// TIA Portal project "双流水线程序控制" (V16)

(* hardware
DEVICE "S7-1200 station_1"  S7-1200 Station
   slot 0: "Rack_0"  S7-1200 Rack  Rack  V1.0
   slot 1: "PLC_1"  CPU 1214C DC/DC/Rly  6ES7 214-1HG40-0XB0  V4.4
*)

// ===== PLC "PLC_1"  CPU 1214C DC/DC/Rly =====

VAR_GLOBAL   // PLC tag table "默认变量表"
   "Tag_1" AT %M1.0 : Bool;
   "Tag_2" AT %M1.1 : Bool;
END_VAR

VAR_GLOBAL   // PLC tag table "io表"
   "传感器9" AT %I0.0 : Bool;
   "传感器8" AT %I0.1 : Bool;
   "传感器7" AT %I0.2 : Bool;
   "传感器1" AT %I0.3 : Bool;
   "传感器2" AT %I0.4 : Bool;
   "传感器3" AT %I0.5 : Bool;
   "传感器4" AT %I0.6 : Bool;
   "传感器5" AT %I0.7 : Bool;
   "传感器6" AT %I1.0 : Bool;
   "传感器10" AT %I1.1 : Bool;
   "开始" AT %I1.2 : Bool;
   "复位" AT %I1.3 : Bool;
   "停止" AT %I1.4 : Bool;
   "紧急停止" AT %I1.5 : Bool;
   "1挡" AT %I1.6 : Bool;
   "FACTORY I/O (Running)" AT %I1.7 : Bool;
   "前后" AT %Q0.0 : Bool;
   "上下" AT %Q0.1 : Bool;
   "吸取" AT %Q0.2 : Bool;
   "皮带1" AT %Q0.3 : Bool;
   "推上盖" AT %Q0.4 : Bool;
   "上升1" AT %Q0.5 : Bool;
   "皮带2" AT %Q0.6 : Bool;
   "推下盖" AT %Q0.7 : Bool;
   "上升2" AT %Q1.0 : Bool;
   "绿灯" AT %Q1.1 : Bool;
   "黄灯" AT %Q1.2 : Bool;
   "红灯" AT %Q1.3 : Bool;
   "显示屏" AT %QD30 : DInt;
END_VAR

// folder: 02-启动

DATA_BLOCK "启动_DB"   // DB2
{ S7_Optimized_Access := 'TRUE' }
VERSION : 0.1
// stored: InstanceOfName 启动
"启动"
BEGIN
END_DATA_BLOCK

// folder: 02-核心组装区

DATA_BLOCK "核心组装区_DB"   // DB1
{ S7_Optimized_Access := 'TRUE' }
VERSION : 0.1
// stored: InstanceOfName 核心组装区
"核心组装区"
BEGIN
END_DATA_BLOCK

// folder: (top level)

FUNCTION "MHJ-PLC-Lab-Function-S71200" : Void   // FC9000, SCL
{ S7_Optimized_Access := 'TRUE' }
VERSION : 0.1
   VAR_TEMP
      rdTimeReturn : Int;
      outputTime : DTL;
      SyncVal : Byte;
      forVal : Int;
      forVal_2 : Int;
      Value : Byte;
   END_VAR
   VAR CONSTANT
      CompVal : Byte := 16#34;
      Value_01 : Byte := 16#11;
      Value_01_DW : DWord := 16#A165_D992;
      Value_02_DW : DWord := 16#58BE_4401;
   END_VAR
BEGIN

   #Value:=PEEK(area := 16#82,
        dbNumber := 0,
        byteOffset := 511);
   #Value := #Value + 1;

   POKE(area := 16#82,
        dbNumber := 0,
        byteOffset := 511,
        value := #Value);

   POKE(area:=16#81,
        dbNumber:=0,
        byteOffset:=1016,
        value:=#Value_01_DW);
   POKE(area := 16#81,
        dbNumber := 0,
        byteOffset := 1020,
        value := #Value_02_DW);

   POKE(area := 16#81,
        dbNumber := 0,
        byteOffset := 511,
        value := B#16#00);

   FOR #forVal := 0 TO 120 DO
       FOR #forVal_2:=0 TO 10 DO
           #rdTimeReturn:=RD_SYS_T(#outputTime);
           #rdTimeReturn := WR_SYS_T(#outputTime);
           #rdTimeReturn := RD_SYS_T(#outputTime);
           #rdTimeReturn := WR_SYS_T(#outputTime);
       END_FOR;
       #SyncVal:= PEEK(area := 16#81,
                      dbNumber := 0,
                      byteOffset := 511);
       IF #SyncVal = #CompVal THEN
          GOTO M_1;
       END_IF;
   END_FOR;
   RETURN;

   M_1:
   POKE(area := 16#81,
        dbNumber := 0,
        byteOffset := 511,
        value := B#16#0);
END_FUNCTION

ORGANIZATION_BLOCK "Main"   // OB1, LAD, ProgramCycle
TITLE = "Main Program Sweep (Cycle)"
{ S7_Optimized_Access := 'TRUE' }
VERSION : 0.1
   VAR_INPUT
      Initial_Call : Bool;   // Initial call of this OB
      Remanence : Bool;   // =True, if remanent data are available
   END_VAR
BEGIN

REGION Network 1
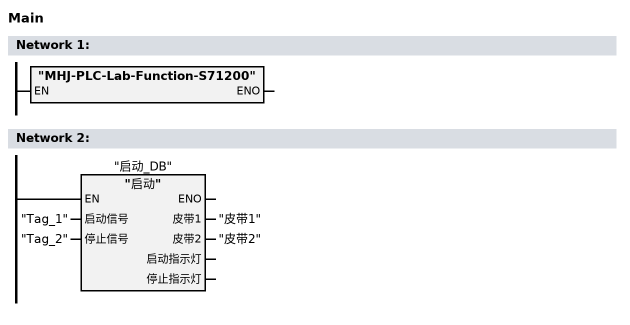
   RUNG wire#powerrail
      "MHJ-PLC-Lab-Function-S71200"()
   END_RUNG
   // the same network as SCL:
   "MHJ-PLC-Lab-Function-S71200"();
END_REGION

REGION Network 2
   RUNG wire#powerrail
      "启动_DB"(启动信号 := "Tag_1", 停止信号 := "Tag_2", 皮带1 => "皮带1", 皮带2 => "皮带2", 启动指示灯 =>, 停止指示灯 =>)
   END_RUNG
   // the same network as SCL:
   "启动_DB"(启动信号 := "Tag_1", 停止信号 := "Tag_2", 皮带1 => "皮带1", 皮带2 => "皮带2");   // "启动"
END_REGION
END_ORGANIZATION_BLOCK

// folder: 01-初始化

FUNCTION_BLOCK "初始化"   // FB1, LAD
{ S7_Optimized_Access := 'TRUE' }
VERSION : 0.1
BEGIN
END_FUNCTION_BLOCK

// folder: 02-启动

FUNCTION_BLOCK "启动"   // FB3, LAD
{ S7_Optimized_Access := 'TRUE' }
VERSION : 0.1
   VAR_INPUT
      启动信号 : Bool;
      停止信号 : Bool;
   END_VAR
   VAR_OUTPUT
      皮带1 : Bool;
      皮带2 : Bool;
      启动指示灯 : Bool;
      停止指示灯 : Bool;
   END_VAR
BEGIN

REGION Network 1
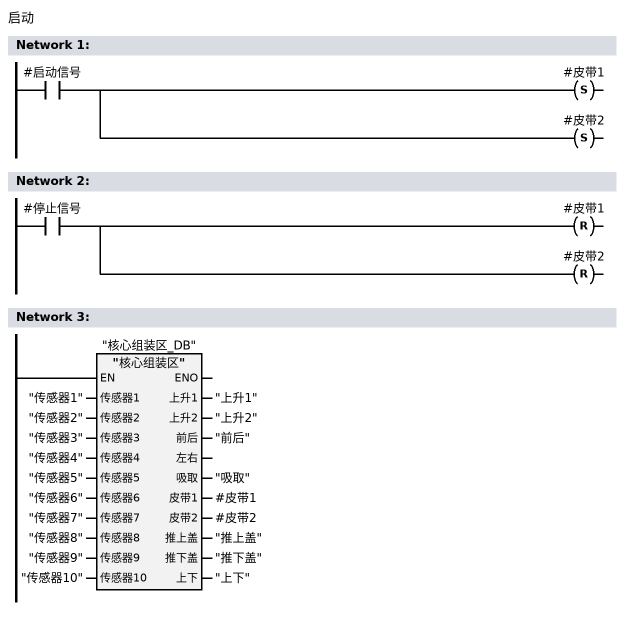
   RUNG wire#powerrail
      Contact( #启动信号 )
      wire#w1
      S_Coil( #皮带1 )
   END_RUNG
   RUNG wire#w1
      S_Coil( #皮带2 )
   END_RUNG
   // the same network as SCL:
   IF #启动信号 THEN
       #皮带1 := TRUE;
       #皮带2 := TRUE;
   END_IF;
END_REGION

REGION Network 2
   RUNG wire#powerrail
      Contact( #停止信号 )
      wire#w1
      R_Coil( #皮带1 )
   END_RUNG
   RUNG wire#w1
      R_Coil( #皮带2 )
   END_RUNG
   // the same network as SCL:
   IF #停止信号 THEN
       #皮带1 := FALSE;
       #皮带2 := FALSE;
   END_IF;
END_REGION

REGION Network 3
   RUNG wire#powerrail
      "核心组装区_DB"(传感器1 := "传感器1", 传感器2 := "传感器2", 传感器3 := "传感器3", 传感器4 := "传感器4", 传感器5 := "传感器5", 传感器6 := "传感器6", 传感器7 := "传感器7", 传感器8 := "传感器8", 传感器9 := "传感器9", 传感器10 := "传感器10", 上升1 => "上升1", 上升2 => "上升2", 前后 => "前后", 左右 =>, 吸取 => "吸取", 皮带1 => #皮带1, 皮带2 => #皮带2, 推上盖 => "推上盖", 推下盖 => "推下盖", 上下 => "上下")
   END_RUNG
   // the same network as SCL:
   "核心组装区_DB"(传感器1 := "传感器1",   // "核心组装区"
              传感器2 := "传感器2",
              传感器3 := "传感器3",
              传感器4 := "传感器4",
              传感器5 := "传感器5",
              传感器6 := "传感器6",
              传感器7 := "传感器7",
              传感器8 := "传感器8",
              传感器9 := "传感器9",
              传感器10 := "传感器10",
              上升1 => "上升1",
              上升2 => "上升2",
              前后 => "前后",
              吸取 => "吸取",
              皮带1 => #皮带1,
              皮带2 => #皮带2,
              推上盖 => "推上盖",
              推下盖 => "推下盖",
              上下 => "上下");
END_REGION
END_FUNCTION_BLOCK

// folder: 02-核心组装区

FUNCTION_BLOCK "核心组装区"   // FB2, LAD
{ S7_Optimized_Access := 'TRUE' }
VERSION : 0.1
   VAR_INPUT
      传感器1 : Bool;
      传感器2 : Bool;
      传感器3 : Bool;
      传感器4 : Bool;
      传感器5 : Bool;
      传感器6 : Bool;
      传感器7 : Bool;
      传感器8 : Bool;
      传感器9 : Bool;
      传感器10 : Bool;
   END_VAR
   VAR_OUTPUT
      上升1 : Bool;
      上升2 : Bool;
      前后 : Bool;
      左右 : Bool;
      吸取 : Bool;
      皮带1 : Bool;
      皮带2 : Bool;
      推上盖 : Bool;
      推下盖 : Bool;
      上下 : Bool;
   END_VAR
   VAR
      吸附准备 : Bool;
      IEC_Timer_0_Instance : TON_TIME;
      上下复位 : Bool;
      IEC_Timer_0_Instance_1 : TON_TIME;
      上升2准备 : Bool;
      中间变量1 : Bool;
      中间变量2 : Bool;
      中间变量3 : Bool;
      中间变量4 : Bool;
      中间变量5 : Bool;
      中间变量6 : Bool;
      中间变量7 : Bool;
      中间变量8 : Bool;
      中间变量9 : Bool;
      中间变量10 : Bool;
      中间变量11 : Bool;
      中间变量12 : Bool;
      中间变量13 : Bool;
      中间变量14 : Bool;
   END_VAR
   VAR_TEMP   // added for the SCL form of the ladder/FBD networks
      _w1 : Bool;
      _w2 : Bool;
      _w3 : Bool;
      _w4 : Bool;
   END_VAR
BEGIN

REGION Network 1: 关闭传送带，启动推杆
   // 因为传感器常开，当感应到物体之后，到物体离开形成一个下降沿，为了避免上升2还没有回归就开始推
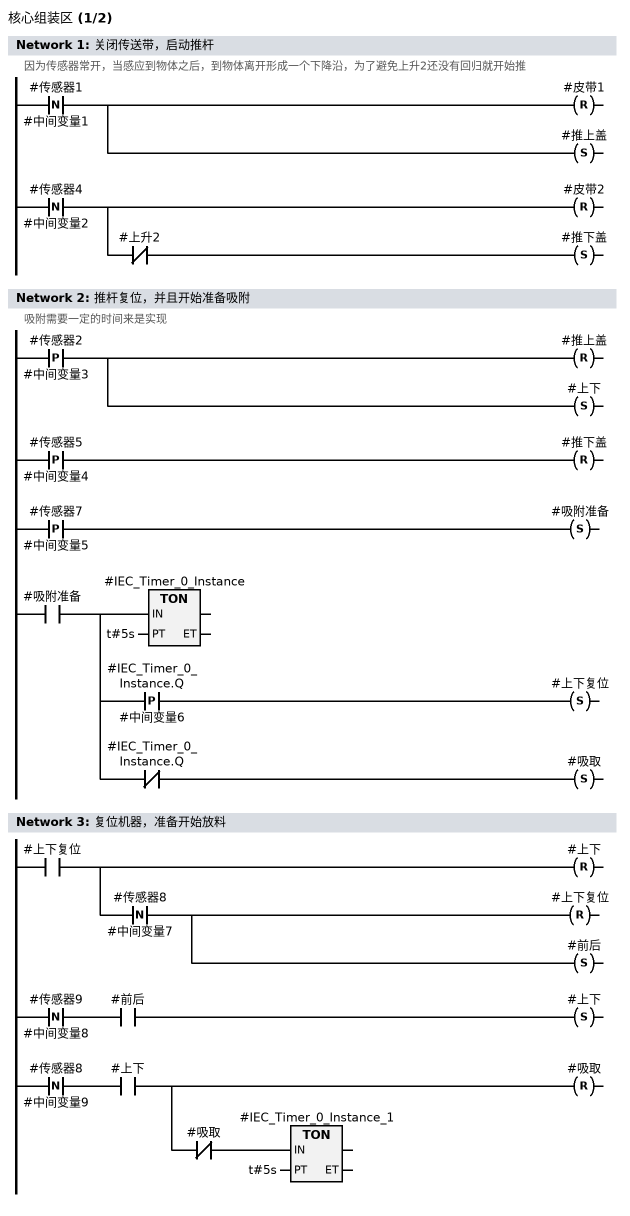
   RUNG wire#powerrail
      N_Contact(operand := #传感器1, bit := #中间变量1)
      wire#w1
      R_Coil( #皮带1 )
   END_RUNG
   RUNG wire#w1
      S_Coil( #推上盖 )
   END_RUNG
   RUNG wire#powerrail
      N_Contact(operand := #传感器4, bit := #中间变量2)
      wire#w2
      R_Coil( #皮带2 )
   END_RUNG
   RUNG wire#w2
      I_Contact( #上升2 )
      S_Coil( #推下盖 )
   END_RUNG
   // the same network as SCL:
   #_w1 := NOT #传感器1 AND #中间变量1;   // falling edge of #传感器1
   #中间变量1 := #传感器1;
   IF #_w1 THEN
       #皮带1 := FALSE;
       #推上盖 := TRUE;
   END_IF;
   #_w2 := NOT #传感器4 AND #中间变量2;   // falling edge of #传感器4
   #中间变量2 := #传感器4;
   IF #_w2 THEN #皮带2 := FALSE; END_IF;
   IF #_w2 AND NOT #上升2 THEN #推下盖 := TRUE; END_IF;
END_REGION

REGION Network 2: 推杆复位，并且开始准备吸附
   // 吸附需要一定的时间来是实现
   #_w1 := #传感器2 AND NOT #中间变量3;   // rising edge of #传感器2
   #中间变量3 := #传感器2;
   IF #_w1 THEN
       #推上盖 := FALSE;
       #上下 := TRUE;
   END_IF;
   #_w2 := #传感器5 AND NOT #中间变量4;   // rising edge of #传感器5
   #中间变量4 := #传感器5;
   IF #_w2 THEN #推下盖 := FALSE; END_IF;
   #_w3 := #传感器7 AND NOT #中间变量5;   // rising edge of #传感器7
   #中间变量5 := #传感器7;
   IF #_w3 THEN #吸附准备 := TRUE; END_IF;
   #IEC_Timer_0_Instance(IN := #吸附准备, PT := t#5s);   // TON
   #_w4 := #吸附准备 AND #IEC_Timer_0_Instance.Q AND NOT #中间变量6;   // rising edge of #IEC_Timer_0_Instance.Q
   #中间变量6 := #IEC_Timer_0_Instance.Q;
   IF #_w4 THEN #上下复位 := TRUE; END_IF;
   IF #吸附准备 AND NOT #IEC_Timer_0_Instance.Q THEN #吸取 := TRUE; END_IF;
END_REGION

REGION Network 3: 复位机器，准备开始放料
   IF #上下复位 THEN #上下 := FALSE; END_IF;
   #_w1 := #上下复位 AND NOT #传感器8 AND #中间变量7;   // falling edge of #传感器8
   #中间变量7 := #传感器8;
   IF #_w1 THEN
       #上下复位 := FALSE;
       #前后 := TRUE;
   END_IF;
   #_w2 := NOT #传感器9 AND #中间变量8;   // falling edge of #传感器9
   #中间变量8 := #传感器9;
   IF #_w2 AND #前后 THEN #上下 := TRUE; END_IF;
   #_w3 := NOT #传感器8 AND #中间变量9;   // falling edge of #传感器8
   #中间变量9 := #传感器8;
   #_w4 := #_w3 AND #上下;
   IF #_w4 THEN #吸取 := FALSE; END_IF;
   #IEC_Timer_0_Instance_1(IN := #_w4 AND NOT #吸取, PT := t#5s);   // TON
END_REGION

REGION Network 4: 上升，准备传送
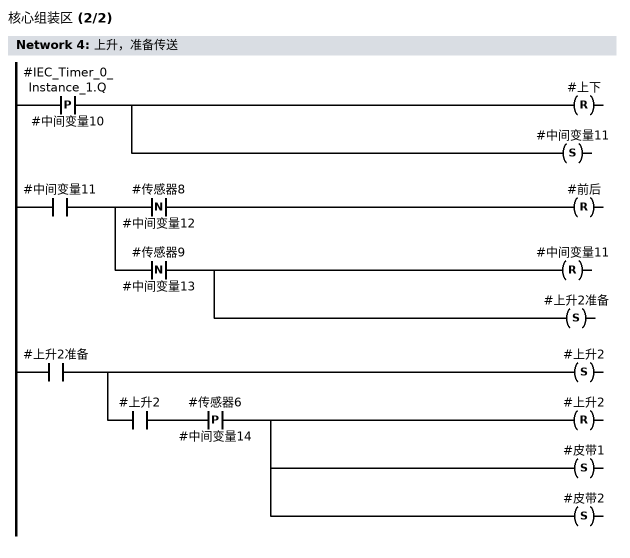
   RUNG wire#powerrail
      P_Contact(operand := #IEC_Timer_0_Instance_1.Q, bit := #中间变量10)
      wire#w1
      R_Coil( #上下 )
   END_RUNG
   RUNG wire#w1
      S_Coil( #中间变量11 )
   END_RUNG
   RUNG wire#powerrail
      Contact( #中间变量11 )
      wire#w2
      N_Contact(operand := #传感器8, bit := #中间变量12)
      R_Coil( #前后 )
   END_RUNG
   RUNG wire#w2
      N_Contact(operand := #传感器9, bit := #中间变量13)
      wire#w3
      R_Coil( #中间变量11 )
   END_RUNG
   RUNG wire#w3
      S_Coil( #上升2准备 )
   END_RUNG
   RUNG wire#powerrail
      Contact( #上升2准备 )
      wire#w4
      S_Coil( #上升2 )
   END_RUNG
   RUNG wire#w4
      Contact( #上升2 )
      P_Contact(operand := #传感器6, bit := #中间变量14)
      wire#w5
      R_Coil( #上升2 )
   END_RUNG
   RUNG wire#w5
      S_Coil( #皮带1 )
   END_RUNG
   RUNG wire#w5
      S_Coil( #皮带2 )
   END_RUNG
   // the same network as SCL:
   #_w1 := #IEC_Timer_0_Instance_1.Q AND NOT #中间变量10;   // rising edge of #IEC_Timer_0_Instance_1.Q
   #中间变量10 := #IEC_Timer_0_Instance_1.Q;
   IF #_w1 THEN
       #上下 := FALSE;
       #中间变量11 := TRUE;
   END_IF;
   #_w2 := #中间变量11 AND NOT #传感器8 AND #中间变量12;   // falling edge of #传感器8
   #中间变量12 := #传感器8;
   IF #_w2 THEN #前后 := FALSE; END_IF;
   #_w3 := #中间变量11 AND NOT #传感器9 AND #中间变量13;   // falling edge of #传感器9
   #中间变量13 := #传感器9;
   IF #_w3 THEN
       #中间变量11 := FALSE;
       #上升2准备 := TRUE;
   END_IF;
   IF #上升2准备 THEN #上升2 := TRUE; END_IF;
   #_w4 := #上升2准备 AND #上升2 AND #传感器6 AND NOT #中间变量14;   // rising edge of #传感器6
   #中间变量14 := #传感器6;
   IF #_w4 THEN
       #上升2 := FALSE;
       #皮带1 := TRUE;
       #皮带2 := TRUE;
   END_IF;
END_REGION
END_FUNCTION_BLOCK